// TIA Portal V21 export
FUNCTION "fcSafety" : Void   // FC1, LAD
{ S7_Optimized_Access := 'TRUE' }
// stored: SetENOAutomatically false
BEGIN

REGION Network 1: Safety
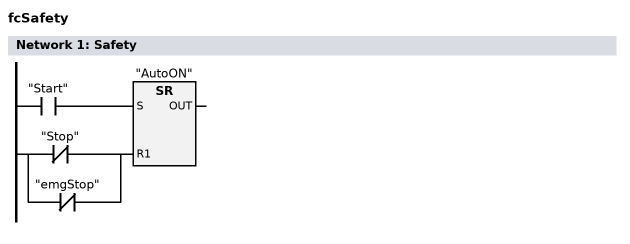
   RUNG wire#powerrail
      Contact( "Start" )
      S_SR(operand := "AutoON", r1 := wire#w1)
   END_RUNG
   RUNG wire#powerrail
      I_Contact( "Stop" )
   END_RUNG wire#w1
   RUNG wire#powerrail
      I_Contact( "emgStop" )
   END_RUNG wire#w1
   // the same network as SCL:
   IF "Start" THEN
       "AutoON" := TRUE;   // SR flip-flop
   END_IF;
   IF NOT "Stop" OR NOT "emgStop" THEN "AutoON" := FALSE; END_IF;
END_REGION
END_FUNCTION
